FUNCTION_BLOCK FB_Spindle
VAR_INPUT
END_VAR
VAR_OUTPUT
END_VAR
VAR
	// ================= Tool Changing ====================================
	pbToolChange AT %I*: BOOL;
	spindleToolLocked AT %I* : BOOL;
	spindleToolOpen AT %I* : BOOL;
	cylinderToolRelease1 AT %Q* : BOOL;
	cylinderToolRelease2 AT %Q* : BOOL;
	spindleClean AT %Q* : BOOL;
	toolChangeTimer : TON;
	tool0 AT %I* : BOOL;
	tool1 AT %I* : BOOL;
	tool2 AT %I* : BOOL;
	tool3 AT %I* : BOOL;
	tool4 AT %I* : BOOL;
	tool5 AT %I* : BOOL;
	tool6 AT %I* : BOOL;
	tool7 AT %I* : BOOL;
	toolLimitSwitchArray : ARRAY[0..8] OF BOOL;
	//Dust Hood
	dustHoodCylinder AT %Q*		: BOOL;
	dustHoodSawActuator AT %Q* : BOOL;
	
	currentTool : Tool_Type := GVL_Programs.noTool;
	toolSelectedAtInitialization : BOOL := FALSE;
	
	//--------------------Spindle TCP communication --------
	fbWriteRegs : FB_MBWriteRegs; //Function call
	fbWriteRegs2 : FB_MBWriteRegs; //Error reset
	fbReadReg	: FB_MBReadRegs; //Drive run/stop
	fbReadReg2	: FB_MBReadRegs; //Error
	fbReadRegSpeed	: FB_MBReadRegs; //Speed
	fbReadRegTorque	: FB_MBReadRegs; //Torque
	ipAddr      : STRING(15) := '192.168.1.5'; //IPADDRESS
	eWriteState	: (WAIT, START, STOP, WRITE); //state machine
	spindleRunStatus : WORD;
	spindleErrorStatus	: WORD;
	spindleTorqueStatus : WORD;
	spindleSpeedStatus	: WORD;
	spindleIsStopped	: BOOL;
	spindleError		: BOOL;
	spindleSpeed		: INT;
	spindleTorque		: INT;
	
	//--------------------Warmup params-----------
	spindleIsWarm 	: BOOL;
	warmupSpeed1 	: INT := 12000;
	warmupTime1 	: TIME := T#240S;
	warmupSpeed2 	: INT := 18000;
	warmupTime2 	: TIME := T#240S;
	warmupSpeed3 	: INT := 24000;
	warmupTime3 	: TIME := T#240S;
	startTime		: TIME;
	elapsedWarmupTime : TIME;
	spindleWarmupOn	: BOOL;
	triggerWarmup	: R_TRIG;
	
	warmUp3: BOOL;
	warmUp2: BOOL;
	warmUp1: BOOL;
	triggerWarm1: R_TRIG;
	triggerWarm2: R_TRIG;
	triggerWarm3: R_TRIG;
	fTrigWarm3 : F_TRIG;
	requestedTool: Tool_Type;
END_VAR

VFD_Status();
//Spindle warmup routine, trigerred from Start_Spindle and stopped with Stop_Spindle
	triggerWarmup(CLK:=spindleWarmupOn);
	triggerWarm1(CLK:=warmUp1);
	triggerWarm2(CLK:=warmUp2);
	triggerWarm3(CLK:=warmUp3);
	fTrigWarm3(CLK := warmUp3);
	
IF spindleWarmupOn THEN
	IF triggerWarmup.Q THEN
		startTime := TIME(); 
	END_IF
		
	elapsedWarmupTime := TIME() - startTime;
	
	IF elapsedWarmupTime > warmUpTime1 + warmupTime2 + warmupTime3 THEN
		warmUp1 := FALSE;
		warmUp2 := FALSE;
		warmUp3 := FALSE;
		Stop_Spindle();
		spindleWarmupOn := FALSE;
		spindleIsWarm := TRUE;
	ELSIF elapsedWarmupTime > warmUpTime1 + warmupTime2 THEN
		warmUp1 := FALSE;
		warmUp2 := FALSE;
		warmUp3 := TRUE;
	ELSIF elapsedWarmupTime > warmUpTime1 THEN
		warmUp1 := FALSE;
		warmUp2 := TRUE;
		warmUp3 := FALSE;
	ELSIF elapsedWarmupTime > T#0S THEN
		warmUp1 := TRUE;
		warmUp2 := FALSE;
		warmUp3 := FALSE;
	END_IF
	
	IF triggerWarm1.Q THEN
		Start_Spindle(spindleSpeed := warmupSpeed1);
	ELSIF triggerWarm2.Q THEN
		Start_Spindle(spindleSpeed := warmupSpeed2);
	ELSIF triggerWarm3.Q THEN
		Start_Spindle(spindleSpeed := warmupSpeed3);
	END_IF

END_IF

METHOD Dust_Hood : BOOL
VAR_INPUT
	x_pose : LREAL;
	enable : BOOL;
END_VAR
IF enable THEN
	IF x_pose < -1060 THEN
		dustHoodCylinder := FALSE;
		dustHoodSawActuator := FALSE;
	ELSE
		dustHoodCylinder := TRUE;
		IF currentTool.toolNumber = 0 THEN
			dustHoodSawActuator := TRUE;
		ELSE
			dustHoodSawActuator := FALSE;
		END_IF
	END_IF
ELSE
	dustHoodCylinder := FALSE;
	dustHoodSawActuator := FALSE;
END_IF
END_METHOD

//Sets tool change cylinders to closed, returns true if tool locked
METHOD Grab_Tool : BOOL 
VAR_INPUT
END_VAR
cylinderToolRelease1 := FALSE;
cylinderToolRelease2 := FALSE;
Grab_Tool := spindleToolLocked;
END_METHOD

METHOD Manual_Tool_Change
VAR_INPUT
	changeToolEnable : BOOL;
END_VAR
IF changeToolEnable THEN
	toolChangeTimer(IN:= pbToolChange, PT:=T#2S);
	
	IF pbToolChange THEN
		IF toolChangeTimer.Q AND spindleIsStopped THEN
			cylinderToolRelease1 := TRUE;
			cylinderToolRelease2 := TRUE;
		END_IF
	ELSE
		cylinderToolRelease1 := FALSE;
		cylinderToolRelease2 := FALSE;
	END_IF
END_IF
END_METHOD

METHOD Release_Tool : BOOL; //Sets tool change cylinders to open, returns true if tool released
VAR_INPUT
END_VAR
IF spindleIsStopped THEN
	cylinderToolRelease1 := TRUE;
	cylinderToolRelease2 := TRUE;
	Release_Tool := spindleToolOpen;
ELSE
	cylinderToolRelease1 := FALSE;
	cylinderToolRelease2 := FALSE;
	Release_Tool := FALSE;
END_IF
END_METHOD

//Resets drive, returns true if no drive error
METHOD Reset_Drive : BOOL
VAR_INPUT
END_VAR
VAR
	errorReset : WORD := INT_TO_WORD(2);
END_VAR
fbWriteRegs2(
			sIPAddr:= ipAddr, 
			nTCPPort:= 502, 
			nUnitID:= 16#FF, 
			nQuantity:= 1, 
			nMBAddr:= 16#2002, 
			cbLength:= SIZEOF(errorReset), 
			pSrcAddr:= ADR(errorReset), 
			bExecute:= FALSE, 
			tTimeout:= , 
			bBusy=> , 
			bError=> , 
			nErrId=> );
			
fbWriteRegs2(
			sIPAddr:= ipAddr, 
			nTCPPort:= 502, 
			nUnitID:= 16#FF, 
			nQuantity:= 1, 
			nMBAddr:= 16#2002, 
			cbLength:= SIZEOF(errorReset), 
			pSrcAddr:= ADR(errorReset), 
			bExecute:= TRUE, 
			tTimeout:= , 
			bBusy=> , 
			bError=> , 
			nErrId=> );
			
IF NOT spindleError THEN
	Reset_Drive := TRUE;
END_IF
END_METHOD

//Starts spindle warmup, called in fbSpindle
METHOD Spindle_Warmup
VAR_INPUT
END_VAR
spindleWarmupOn := TRUE;
END_METHOD

//Description:
//This method is responsible for starting the spindle motor based on the input speed provided in revolutions per minute (RPM). It converts the spindle speed into frequency and initiates the spindle motor accordingly.

//Parameters:
//- spindleSpeed: INT - The desired spindle speed in RPM.

//Returns:
//This method does not return any value.
METHOD Start_Spindle
VAR_INPUT
	spindleSpeed : INT; //Spindle speed RPM
	
END_VAR

VAR
	spindleFrequency : INT := (spindleSpeed - 12000) / 30 + 400; //Speed conversion to frequency
	startValue  : ARRAY [0..1] OF WORD := [INT_TO_WORD(18), INT_TO_WORD(SpindleFrequency*10)];
END_VAR
fbWriteRegs(
			sIPAddr:= ipAddr, 
			nTCPPort:= 502, 
			nUnitID:= 16#FF, 
			nQuantity:= 2, 
			nMBAddr:= 16#2000, 
			cbLength:= SIZEOF(startValue), 
			pSrcAddr:= ADR(startValue), 
			bExecute:= FALSE, 
			tTimeout:= , 
			bBusy=> , 
			bError=> , 
			nErrId=> );
			
fbWriteRegs(
			sIPAddr:= ipAddr, 
			nTCPPort:= 502, 
			nUnitID:= 16#FF, 
			nQuantity:= 2, 
			nMBAddr:= 16#2000, 
			cbLength:= SIZEOF(startValue), 
			pSrcAddr:= ADR(startValue), 
			bExecute:= TRUE, 
			tTimeout:= , 
			bBusy=> , 
			bError=> , 
			nErrId=> );
			
spindleClean := TRUE;
END_METHOD

//Stops spindle
METHOD Stop_Spindle
VAR_INPUT
END_VAR

VAR
	stopValue: ARRAY [0..1] OF WORD := [INT_TO_WORD(1), INT_TO_WORD(0)];
END_VAR
fbWriteRegs(
			sIPAddr:= ipAddr, 
			nTCPPort:= 502, 
			nUnitID:= 16#FF, 
			nQuantity:= 2, 
			nMBAddr:= 16#2000, 
			cbLength:= SIZEOF(stopValue), 
			pSrcAddr:= ADR(stopValue), 
			bExecute:= FALSE, 
			tTimeout:= , 
			bBusy=> , 
			bError=> , 
			nErrId=> );

fbWriteRegs(
			sIPAddr:= ipAddr, 
			nTCPPort:= 502, 
			nUnitID:= 16#FF, 
			nQuantity:= 2, 
			nMBAddr:= 16#2000, 
			cbLength:= SIZEOF(stopValue), 
			pSrcAddr:= ADR(stopValue), 
			bExecute:= TRUE, 
			tTimeout:= , 
			bBusy=> , 
			bError=> , 
			nErrId=> );
			
spindleWarmupOn := FALSE;
warmup1 := FALSE;
warmup2 := FALSE;
warmup3 := FALSE;
spindleClean := FALSE;
END_METHOD

//Updates the current tool based on an integer
METHOD Update_Current_Tool : BOOL
VAR_INPUT
	toolNumber : INT;
END_VAR
VAR
	updatedTool : Tool_Type;
	success : BOOL;
END_VAR
success := TRUE;
CASE toolNumber OF
		0:
			updatedTool := GVL_Programs.sawblade;
		6:
			updatedTool := GVL_Programs.halfInchBall;
		2:
			updatedTool := GVL_Programs.quarterInchUpcut;
		5:
			updatedTool := GVL_Programs.dovetail;
		4:
			updatedTool := GVL_Programs.halfInchUpcut;
		8:
			updatedTool := GVL_Programs.noTool;
			
		ELSE
			success := FALSE;
	END_CASE
		
currentTool := updatedTool;
	
// Successfully updated the current tool
IF NOT success THEN
	Update_Current_Tool := FALSE;
ELSE
	Update_Current_Tool := TRUE;
	toolSelectedAtInitialization := TRUE;
END_IF
END_METHOD

METHOD Update_Requested_Tool : BOOL
VAR_INPUT
	toolNumber : INT;
END_VAR
VAR
	updatedTool : Tool_Type;
	success : BOOL;
END_VAR
CASE toolNumber OF
		0:
			updatedTool := GVL_Programs.sawblade;
		6:
			updatedTool := GVL_Programs.halfInchBall;
		2:
			updatedTool := GVL_Programs.quarterInchUpcut;
		5:
			updatedTool := GVL_Programs.dovetail;
		4:
			updatedTool := GVL_Programs.halfInchUpcut;
		8:
			updatedTool := GVL_Programs.noTool;
			
		ELSE
			success := FALSE;
	END_CASE
		
requestedTool := updatedTool;
	
// Successfully updated the current tool
IF NOT success THEN
	Update_Requested_Tool := FALSE;
ELSE
	Update_Requested_Tool := TRUE;
END_IF
END_METHOD

METHOD Verify_Tool_Change_Request : BOOL
VAR_INPUT
	toolToDrop : UINT;
	toolToPickup : UINT;
END_VAR
//NC contacts. Detect if current tool holder is empty and requested tool holder is full. If no tool is selected as dropoff, checks if all other slots are full.
toolLimitSwitchArray[0] := tool0;
toolLimitSwitchArray[1] := tool1;
toolLimitSwitchArray[2] := tool2;
toolLimitSwitchArray[3] := tool3;
toolLimitSwitchArray[4] := tool4;
toolLimitSwitchArray[5] := tool5;
toolLimitSwitchArray[6] := tool6;
toolLimitSwitchArray[7] := tool7;

IF (toolLimitSwitchArray[toolToDrop] OR (toolToDrop = 8 AND NOT toolLimitSwitchArray[0] AND NOT toolLimitSwitchArray[2] AND NOT toolLimitSwitchArray[4])) AND (NOT toolLimitSwitchArray[toolToPickup] OR toolToPickup = 8) OR (toolToDrop = toolToPickup AND toolLimitSwitchArray[toolToDrop]) THEN 
	Verify_Tool_Change_Request := TRUE;
ELSE
	Verify_Tool_Change_Request := FALSE;
END_IF
//Verify_Tool_Change_Request := TRUE; //TODO: remove once wired!!
END_METHOD

//Updates the status of the VFD: whether it's stopped and whether it is in error state
METHOD VFD_Status : BOOL //returns true if drive has no error
VAR_INPUT
END_VAR
VAR
	runStatus : USINT;
	errorStatus : USINT;
END_VAR
fbReadReg(
			sIPAddr:= ipAddr, 
			nTCPPort:= 502, 
			nUnitID:= 16#FF, 
			nQuantity:= 1, 
			nMBAddr:= 16#2101, 
			cbLength:= SIZEOF(spindleRunStatus), 
			pDestAddr := ADR(spindleRunStatus), 
			bExecute:= FALSE, 
			tTimeout:= , 
			bBusy=> , 
			bError=> , 
			nErrId=> );
			
fbReadReg(
			sIPAddr:= ipAddr, 
			nTCPPort:= 502, 
			nUnitID:= 16#FF, 
			nQuantity:= 1, 
			nMBAddr:= 16#2101, 
			cbLength:= SIZEOF(spindleRunStatus), 
			pDestAddr := ADR(spindleRunStatus), 
			bExecute:= TRUE, 
			tTimeout:= , 
			bBusy=> , 
			bError=> , 
			nErrId=> );
			
fbReadReg2(
			sIPAddr:= ipAddr, 
			nTCPPort:= 502, 
			nUnitID:= 16#FF, 
			nQuantity:= 1, 
			nMBAddr:= 16#2226, 
			cbLength:= SIZEOF(spindleErrorStatus), 
			pDestAddr := ADR(spindleErrorStatus), 
			bExecute:= FALSE, 
			tTimeout:= , 
			bBusy=> , 
			bError=> , 
			nErrId=> );

fbReadReg2(
			sIPAddr:= ipAddr, 
			nTCPPort:= 502, 
			nUnitID:= 16#FF, 
			nQuantity:= 1, 
			nMBAddr:= 16#2226, 
			cbLength:= SIZEOF(spindleErrorStatus), 
			pDestAddr := ADR(spindleErrorStatus), 
			bExecute:= TRUE, 
			tTimeout:= , 
			bBusy=> , 
			bError=> , 
			nErrId=> );
			
fbReadRegSpeed(
			sIPAddr:= ipAddr, 
			nTCPPort:= 502, 
			nUnitID:= 16#FF, 
			nQuantity:= 1, 
			nMBAddr:= 16#210C, 
			cbLength:= SIZEOF(spindleSpeedStatus), 
			pDestAddr := ADR(spindleSpeedStatus), 
			bExecute:= FALSE, 
			tTimeout:= , 
			bBusy=> , 
			bError=> , 
			nErrId=> );

fbReadRegSpeed(
			sIPAddr:= ipAddr, 
			nTCPPort:= 502, 
			nUnitID:= 16#FF, 
			nQuantity:= 1, 
			nMBAddr:= 16#210C, 
			cbLength:= SIZEOF(spindleSpeedStatus), 
			pDestAddr := ADR(spindleSpeedStatus), 
			bExecute:= TRUE, 
			tTimeout:= , 
			bBusy=> , 
			bError=> , 
			nErrId=> );
			
fbReadRegTorque(
			sIPAddr:= ipAddr, 
			nTCPPort:= 502, 
			nUnitID:= 16#FF, 
			nQuantity:= 1, 
			nMBAddr:= 16#210B, 
			cbLength:= SIZEOF(spindleTorqueStatus), 
			pDestAddr := ADR(spindleTorqueStatus), 
			bExecute:= FALSE, 
			tTimeout:= , 
			bBusy=> , 
			bError=> , 
			nErrId=> );
fbReadRegTorque(
			sIPAddr:= ipAddr, 
			nTCPPort:= 502, 
			nUnitID:= 16#FF, 
			nQuantity:= 1, 
			nMBAddr:= 16#210B, 
			cbLength:= SIZEOF(spindleTorqueStatus), 
			pDestAddr := ADR(spindleTorqueStatus), 
			bExecute:= TRUE, 
			tTimeout:= , 
			bBusy=> , 
			bError=> , 
			nErrId=> );

runStatus := WORD_TO_USINT(spindleRunStatus);
IF runStatus.0 = 0 AND runStatus.1 = 0 THEN
	spindleIsStopped := TRUE;
ELSE 
	spindleIsStopped := FALSE;
END_IF

errorStatus := WORD_TO_USINT(spindleErrorStatus);
IF errorStatus.3 = 1 AND errorStatus.2 = 0 THEN
	spindleError := TRUE;
ELSE 
	spindleError := FALSE;
END_IF

spindleSpeed := WORD_TO_INT(SpindleSpeedStatus);
spindleTorque := WORD_TO_INT(SpindleTorqueStatus);

VFD_Status := NOT spindleError;
END_METHOD

END_FUNCTION_BLOCK

(* stored: Version 1.1.0.1, ProductVersion 3.1.4024.12
   POU FB_Spindle: Id {3dc147eb-3dde-4052-8db8-ee0200a73c1f}, SpecialFunc None
   Method Dust_Hood: Id {75eb1e7d-7e88-4ff3-acdf-1fc2cf420d06}
   Method Grab_Tool: Id {b157a71e-63d7-43c6-8cda-129fe8943333}
   Method Manual_Tool_Change: Id {caf02692-220f-45ea-9a62-11b6af7ca524}
   Method Release_Tool: Id {44458576-a982-4dd8-917f-a23f3b30cecf}
   Method Reset_Drive: Id {9a8ab2d1-8aed-4c9c-967c-6e187f19fbf4}
   Method Spindle_Warmup: Id {6626f887-e6c9-4081-bd79-0ba0a3b91bcb}
   Method Start_Spindle: Id {702c570c-7182-409d-ac49-a3e78d7a4915}
   Method Stop_Spindle: Id {ef644fdc-e119-4b63-a532-fadf07840f86}
   Method Update_Current_Tool: Id {d316eb47-28e5-4b11-bbfd-0a31ae49903c}
   Method Update_Requested_Tool: Id {85d5d331-1534-446d-a912-cbacd40c27a7}
   Method Verify_Tool_Change_Request: Id {93de9ffd-c991-4212-b109-f473dd00ac57}
   Method VFD_Status: Id {3c5755fa-2782-4792-9f43-a3613d83a04f} *)
